(* IEC 61131-3 sources: ST/projects/struct-array, 2 files *)

(* ---- struct-motor.st ---- *)
TYPE motor :
STRUCT
	manuel_start    :BOOL;
	automatic_start :BOOL;
	stop            :BOOL;
	reset           :BOOL;
END_STRUCT
END_TYPE

(* ---- project.st ---- *)
PROGRAM PLC_PRG
VAR
	motors : ARRAY[1..10] OF motor;
END_VAR

IF motors[3].manuel_start = TRUE AND motors[2].manuel_start THEN
	motors[5].automatic_start := TRUE;
END_IF

END_PROGRAM
